// TIA Portal V17 export
// export: Created 2025-06-26T07:49:16.496631Z, ExportSetting WithDefaults, DisplayName Totally Integrated Automation Portal, DisplayVersion V17 Update 8, DisplayName TIA Portal Openness, DisplayVersion V17 Update 8, DisplayName TIA Portal Version Control Interface, DisplayVersion V17, DisplayName STEP 7 Professional, DisplayVersion V17 Update 8, DisplayName STEP 7 Safety, DisplayVersion V17 Update 6, DisplayName WinCC Advanced, DisplayVersion V17 Update 8
DATA_BLOCK "InputProcessing_DB"   // DB16
AUTHOR : Heaten
VERSION : 0.1
// stored: AutoNumber true, DBAccessibleFromOPCUA true, InstanceOfName InputProcessing, InstanceOfType FB
"InputProcessing"
   // VAR
   //    PumaInputProcessing : "PumaInputProcessing";
   //    CustomerInputProcessing { S7_SetPoint := 'True'} : "CustomerInputProcessing";
   // END_VAR
BEGIN
END_DATA_BLOCK
